// SIMATIC S7-200 SMART project (STEP 7-Micro/WIN SMART), CPU SR40

SYMBOL_TABLE 
USS_LOW_V        VD1000
USS_HIGH_V       VD1004
USS_TIME_OUT     VW1008
USS_I_LINE       VW1010
USS_DAT_PTR0     VD1012
USS_ACT_DRV0     VD1016
USS_CUR_DRV0     VD1020
USS_P0           V1024.0
USS_REQ_SNT0     V1024.1
USS_RETRY_P0     VB1025
USS_ERR_CODE     VB1026
USS_CS_D0        VD1027
USS_CS_W0        VW1027
USS_CS_W2        VW1029
USS_CS_B0        VB1027
USS_CS_B1        VB1028
USS_POLL_BUF     VB1031
USS_XMT_0        VB1046
USS_XMT_ADR0     VB1049
USS_X_STWD       VD1056
USS_X_BCC        VB1060
USS_X_DW1        VD1047
USS_X_DW5        VD1051
USS_X_DW9        VD1055
USS_X_DB13       VB1059
USS_RCV_BUF0     VB1061
USS_R_STX        VB1062
USS_R_LGE        VB1063
USS_R_ADR        VB1064
USS_R_STWD       VD1071
USS_R_DW1        VD1062
USS_R_DW5        VD1066
USS_R_DW9        VD1070
USS_R_W13        VW1074
USS_STAT_TAB     VB1076
USS_ADR_P0       VB1396
END_SYMBOL_TABLE

ORGANIZATION_BLOCK 主:OB1
TITLE=主程序，使用RCV指令和接收完成中断接收数据 
BEGIN
Network 1
// 接收完最大字符数设置的字节时结束报文接收
LD     SM0.1
MOVB   5, SMB130
MOVB   16#DC, SMB187
MOVW   +2, SMW190
MOVB   16#FF, SMB188
MOVW   16, SMW192
MOVB   20, SMB194
ATCH   INT_0:INT0, 24
ATCH   INT_2:INT2, 26
ENI
RCV    VB100, 1
END_ORGANIZATION_BLOCK

SUBROUTINE_BLOCK 异或运算:SBR2
TITLE=
VAR_INPUT
地址指针:DWORD;	// LD0 
字节数B:BYTE;	// LB4 
END_VAR
VAR_OUTPUT
异或结果:BYTE;	// LB5 
END_VAR
VAR
循环计数器:INT;	// LW6 
字节数I:INT;	// LW8 
END_VAR
BEGIN
Network 1
// 网络标题
// 网络注释
LD     SM0.0
MOVB   0, #异或结果:LB5
BTI    #字节数B:LB4, #字节数I:LW8
FOR    #循环计数器:LW6, 1, #字节数I:LW8
Network 2
LD     SM0.0
XORB   *#地址指针:LD0, #异或结果:LB5
INCD   #地址指针:LD0
Network 3
NEXT
END_SUBROUTINE_BLOCK

INTERRUPT_BLOCK INT_0:INT0
TITLE= 接收完成中断程序INT_0
VAR
PNT:DINT;	// LD0 
NUMB:DINT;	// LD4 
SUM1:BYTE;	// LB8 
SUM2:BYTE;	// LB9 
END_VAR
BEGIN
Network 1
// 接收完成中断程序
LD     SM0.0
MOVD   0, #NUMB:LD4
MOVB   VB100, LB7
MOVD   &VB100, #PNT:LD0
+D     #NUMB:LD4, #PNT:LD0
MOVB   *#PNT:LD0, #SUM1:LB8
DECB   LB7
DECB   LB7
CALL   异或运算:SBR2, &VB102, LB7, #SUM2:LB9
?000
Network 2
LDB=   #SUM1:LB8, #SUM2:LB9
R      Q1.0, 1
MOVB   5, SMB34
ATCH   INT_1:INT1, 10
CRETI
NOT
S      Q1.0, 1
RCV    VB100, 1
END_INTERRUPT_BLOCK

INTERRUPT_BLOCK INT_1:INT1
TITLE= 
//  定时中断程序INT_1
BEGIN
Network 1
// 定时中断程序
LD     SM0.0
DTCH   10
XMT    VB100, 1
// 
END_INTERRUPT_BLOCK

INTERRUPT_BLOCK INT_2:INT2
TITLE=发送完成中断程序INT_2
BEGIN
Network 1
// 发送完成中断程序
LD     SM0.0
RCV    VB100, 1
// 
END_INTERRUPT_BLOCK
